FUNCTION WRITE_ANY_DATE_AND_TIME : BOOL
VAR_INPUT
    ptr: POINTER TO DATE_AND_TIME;
    val: DATE_AND_TIME;
END_VAR

ptr^ := val;

END_FUNCTION

(* stored: Version 1.1.0.1, ProductVersion 3.1.4022.9
   POU WRITE_ANY_DATE_AND_TIME: Id {af0064cc-fa42-4eeb-9659-37d82d6b5671}, SpecialFunc None *)
